FUNCTION_BLOCK MultipleChangeDetectVars (* Composite Function Block Type *)
  (* Standard: 61499-2 *)
  (* Version 0.0, 11/1/2016, chivdan, nxtControl GmbH, template *)
  PACKAGE Main;
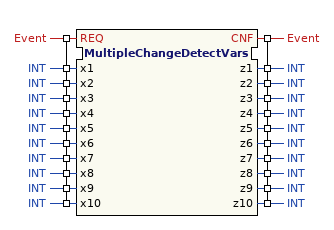
  EVENT_INPUT
    REQ WITH x1, x2, x3, x4, x5, x7, x6, x8, x9, x10; (* Normal Execution Request *)
  END_EVENT
  EVENT_OUTPUT
    CNF WITH z1, z2, z3, z4, z5, z6, z7, z8, z9, z10; (* Execution Confirmation *)
  END_EVENT
  VAR_INPUT
    x1 : INT; (* Input event qualifier *)
    x2 : INT;
    x3 : INT;
    x4 : INT;
    x5 : INT;
    x6 : INT;
    x7 : INT;
    x8 : INT;
    x9 : INT;
    x10 : INT;
  END_VAR
  VAR_OUTPUT
    z1 : INT; (* Output event qualifier *)
    z2 : INT;
    z3 : INT;
    z4 : INT;
    z5 : INT;
    z6 : INT;
    z7 : INT;
    z8 : INT;
    z9 : INT;
    z10 : INT;
  END_VAR
END_FUNCTION_BLOCK
